DEVICE_TYPE RevolutionPi (* Revolution Pi controller *)
  (* Standard: 61499 ITA; Description: Copyright (c) 2024 Monika Wenger This program and the accompanying materials are made available under the terms of the Eclipse Public License 2.0 which is available at https://www.eclipse.org/legal/epl-2.0/ SPDX-License-Identifier: EPL-2.0 *)
  (* Version 3.0, 2024-02-10, Monika Wenger, Initial version *)
  PACKAGE iec61499::system;
  VAR_INPUT
    MGR_ID : WSTRING := "localhost:61499"; (* Device manager socket ID *)
  END_VAR
END_DEVICE_TYPE
